INTERFACE I_LoadController

METHOD GetLoad : REAL
END_METHOD

METHOD RestoreLoad
END_METHOD

METHOD ShedLoad
END_METHOD

END_INTERFACE

(* stored: Version 1.1.0.1, ProductVersion 3.1.4024.16
   Itf I_LoadController: Id {e981e0e8-1158-4350-99c2-3b282e1f6330}
   Method GetLoad: Id {da5a0cb9-01d5-48a7-989d-338eaf769e94}
   Method RestoreLoad: Id {bb633029-8385-4fb5-93a2-e2dbd34f5c0f}
   Method ShedLoad: Id {1cd81629-ac95-4414-8f2a-89c58a5fdf64} *)
